TYPE StationPos :
STRUCT
	EntryPOSX: LREAL;
	EntryPOSY: LREAL;
	Theta: LREAL;
	ExitX: LREAL;
	ExitY: LREAL;
	Taschen: ARRAY[1..3] OF TaschenPos;
END_STRUCT
END_TYPE

(* stored: Version 1.1.0.1, ProductVersion 3.1.4024.11
   DUT StationPos: Id {26fe7703-79e6-46cb-9755-c275e5ec8e8e} *)
